Staubli VAL3: start.pgx

program start()
  local trsf l_trTrsf[3]
  local trsf l_trTrsf1
  local num l_nNum
  local bool l_bBool
begin
  l_trTrsf[0]={0,1,0,0,0,0}
   l_trTrsf[1]={0,0,1,0,0,0}
   l_trTrsf[2]={1,0,0,0,0,0}



  call Circumcircle(l_trTrsf,l_trTrsf1,l_nNum,l_bBool)
  if !l_bBool
    popUpMsg("")
  else
    popUpMsg(toString(".5",l_nNum))
  endIf




end
